{attribute 'OPC.UA.DA.StructuredType':=1}
TYPE ST_QrSkill :
STRUCT
    Control     : ST_SkillControl;
    Status      : stExternalStatus;

    Specific    : ST_QrSkillSpecific;
END_STRUCT
END_TYPE

(* stored: Version 1.1.0.1, ProductVersion 3.1.4026.18
   DUT ST_QrSkill: Id {f1b1c57f-cc8e-4488-9913-03a7cb6d08a7} *)
